Fanuc KAREL source: kb00007.KL

-- PROVISIONAL review KL for V1013-1; original PC SHA256 23a54ee6b7647ee7517bd14b648973919d62bd9122326d7b73c6369afada73ad
-- Incomplete behavior may be omitted. Consult companion uncertainty JSON. Do not deploy.
PROGRAM KB00007
%NOLOCKGROUP
BEGIN
  -- UNRESOLVED_PC offsets 5-28; opcodes 27,22,1C,31,4A
  -- UNRESOLVED_PC offsets 33-37; opcodes 7F
END KB00007
